// TIA Portal V20 export
TYPE "IO_Device_Outputs"
   STRUCT
      Life_Trigger : Bool;
      Emergency_Stop_Release : Bool;
      Trigger_Read_Serial_Number_Entrace_Functional_Test : Bool;
      Trigger_Read_Serial_Number_Exit_Functional_Test : Bool;
      Selected_Voltage_220V : Bool;
      Selected_Voltage_127V : Bool;
      Carousel_Frequency_Inverter_Fail : Bool;
      Conveyor_Belt_Functional_Test_Inverter_Fail : Bool;
   END_STRUCT;
END_TYPE
